FUNCTION_BLOCK FB_ElementCompositionCustomized

;

END_FUNCTION_BLOCK

(* stored: Version 1.1.0.1, ProductVersion 3.1.4024.9
   POU FB_ElementCompositionCustomized: Id {95f3da27-97ba-45f4-bceb-4335121d4a01}, SpecialFunc None *)
